FUNCTION Convert_TOD_TO_UINT : Hresult
VAR_INPUT
	in : TOD;
	out : REFERENCE TO UINT;
END_VAR
VAR
	converted : UINT;
END_VAR

converted := TOD_TO_UINT(in);

IF (UINT_TO_TOD(converted) <> in) THEN
	Convert_TOD_TO_UINT := INCOMPATIBLE;
	RETURN;
END_IF

out := converted;

END_FUNCTION

(* stored: Version 1.1.0.1, ProductVersion 3.1.4024.12
   POU Convert_TOD_TO_UINT: Id {8f9b49df-d564-41f6-86c4-78d348e63e43}, SpecialFunc None *)
